{attribute addProperty BoxType "KL1312"}
{attribute addProperty Id "Channel_1Channel_70B606D100Channel_2Channel_70B606D100"}
{attribute addProperty CRC "3525945802"}
{attribute addProperty SizeInBites "0"}
{attribute addProperty SizeInBytes "0"}
TYPE KL1312_D229A9CA :
STRUCT
	{attribute addProperty Name "Channel_1"}
	Channel_1 : Channel_70B606D1;
	{attribute addProperty Name "Channel_2"}
	Channel_2 : Channel_70B606D1;
END_STRUCT
END_TYPE

(* stored: Version 1.2.0.0, ProductVersion 3.1.4024.9
   DUT KL1312_D229A9CA: Id {b6d5b89f-d7c2-4df1-a128-c2bf0b3f581b} *)
